// TIA Portal V16 export
// export: Created 2021-11-12T13:33:03.9027245Z, ExportSetting WithDefaults, DisplayName Totally Integrated Automation Portal, DisplayVersion V16 Update 3, DisplayName TIA Portal Version Control Interface, DisplayVersion V16 Update 2, DisplayName TIA Portal Openness, DisplayVersion V16 Update 3, DisplayName SINAMICS Startdrive Advanced, DisplayVersion V16 Update 5, DisplayName SINAMICS Startdrive G130, G150, S120, S150, SINAMICS MV, S210, DisplayVersion V16 Update 5, DisplayName SINAMICS Startdrive G110M, G120, G120C, G120D, G120P, G115D, DisplayVersion V16 Update 5, DisplayName STEP 7 Professional, DisplayVersion V16 Update 3, DisplayName STEP 7 Safety, DisplayVersion V16, DisplayName WinCC UA Professional, DisplayVersion V16 Update 3
DATA_BLOCK "STATUS_THM2"   // DB114
{ S7_Optimized_Access := 'TRUE' }
VERSION : 0.1
// stored: AutoNumber true, DBAccessibleFromOPCUA true, IsOnlyStoredInLoadMemory false, IsRetainMemResEnabled false, IsWriteProtectedInAS false, MemoryReserve 100
   VAR
      xxxxx___BinarySensors___xxxxx : Byte;
      xxxxx___BinaryOthers___xxxxx : Byte;
      xxxxx___AnalogueSensors___xxxxx : Byte;
      xxxxx___Drives___xxxxx : Byte;
      xxxxx___MaterialFlow___xxxxx : Byte;
      xxxxx___Other___xxxxx : Byte;
      Device : Struct   // PartCnt treba doplnit do interfejsu
         Specific : "UDT_THM_Status_specific";
         PartCnt : Int;   // PartCnt treba doplnit do interfejsu
      END_STRUCT;
      xxxxx___Alarms___xxxxx : Byte;
      THM : Struct   // From furnace / Sumární porucha z tryskače.
         Main : "UDT_Status_main";
         Specific : "UDT_DI_Mon_Status_specific";
         Error { S7_SetPoint := 'True'} : "UDT_Error01";
      END_STRUCT;
      LiveBit : Struct   // Communication / Chyba komunikace.
         Main : "UDT_Status_main";
         Specific : "UDT_DI_Mon_Status_specific";
         Error { S7_SetPoint := 'True'} : "UDT_Error01";
      END_STRUCT;
      ProdParam : Struct   // Production parameters not changed / Produkční parametry nezměneny.
         Main : "UDT_Status_main";
         Specific : "UDT_DI_Mon_Status_specific";
         Error { S7_SetPoint := 'True'} : "UDT_Error01";
      END_STRUCT;
      xxxxx___ProcessAlarms___xxxxx : Byte;
      BlastingMediumNok : Struct   // Blasting medium not OK / Otryskávací médium NOK
         Main : "UDT_Status_main";
         Specific : "UDT_DI_Mon_Status_specific";
         Error { S7_SetPoint := 'True'} : "UDT_Error01";
      END_STRUCT;
      xxxxx__SafetyAlarms__xxxxx : Byte;
      ES : Struct   // E-stop
         Main : "UDT_Status_main";
         Specific { S7_SetPoint := 'True'} : "UDT_DI_Mon_Status_specific";
         Error { S7_SetPoint := 'True'} : "UDT_Error01";
      END_STRUCT;
   END_VAR
BEGIN
END_DATA_BLOCK
